{attribute 'qualified_only'}
VAR_GLOBAL
	g:BOOL;
END_VAR

(* stored: Version 1.1.0.1, ProductVersion 3.1.4024.6
   GVL GVL: Id {9a10cfea-b729-4436-b68f-1886bcbf2bf1} *)
